FUNCTION FC_CallAtStart_EpochTime : BOOL		// Called from FB_Cyclestart, DO NOT call from your application
												// Stores the EPOCH time to IIN.epochtime

// To be called once/cycle

IING.epochtime := (F_GetSystemTime() / 10000) - IING.EPOCH_CORRECTION;	// System is in 100nseconds -> divide by 10000 for milliseconds

END_FUNCTION

(* stored: Version 1.1.0.1, ProductVersion 3.1.4026.18
   POU FC_CallAtStart_EpochTime: Id {3b4901ee-67eb-4924-9100-6b24c3dec127}, SpecialFunc None *)
